TYPE ST_LinearPumpControllDB :
STRUCT
	sPumpNumber		: STRING(2); 
	sOldPosition	: STRING(8);
	sNewPosition	: STRING(8);
	sUserName		: STRING(64);
	sDateOfChange	: STRING(64);
END_STRUCT
END_TYPE

(* stored: Version 1.1.0.1, ProductVersion 3.1.4024.15
   DUT ST_LinearPumpControllDB: Id {85e5e0ef-6827-4294-ba2b-dd1b164ea562} *)
